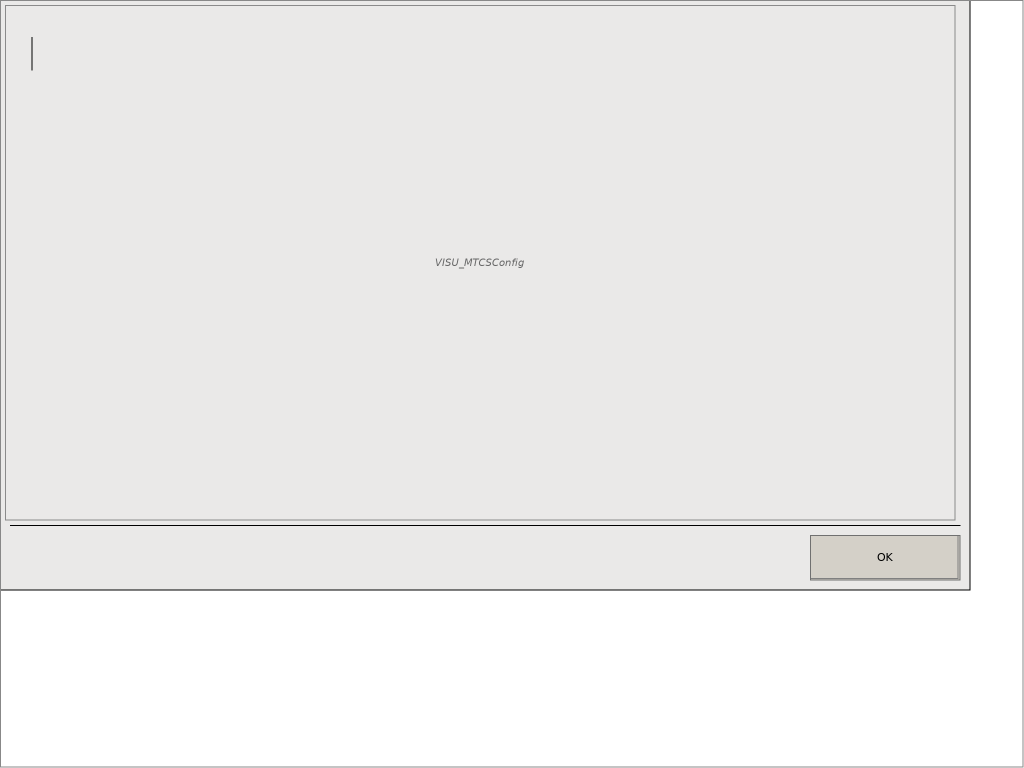
VISUALIZATION VISU_MTCSConfigDialog  // 1024x768
    Rectangle (0,0 970x590)
    Button (810,535 150x45), "OK"
        OnMouseClick: CloseDialog Dialog=VISU_MTCSConfigDialog, Result=OK, NumpadKeypadSet=True
    Line (10,525) (960,525)
    Frame (5,5 950x515)
        shows VISU_MTCSConfig(editableConfig := GLOBAL.mtcs.editableConfig, activeConfig := GLOBAL.mtcs.config, mgr := GLOBAL.mtcs.parts.configManager, mgrWidget := GLOBAL.gui.configManager, widget := GLOBAL.gui)
    Line (32,70) (32,37)
END_VISUALIZATION

(* stored: Version 1.1.0.1, ProductVersion 3.1.4019.2
   Visu VISU_MTCSConfigDialog: Id {d6ed5dff-125f-4ea6-8a24-d8796cea23b9} *)
